TYPE ST_GetCamInfoParams :
STRUCT
  AtMasterPosition  : BOOL;
  MasterPosition    : LREAL;
END_STRUCT
END_TYPE

(* stored: Version 1.1.0.1, ProductVersion 3.1.4023.8
   DUT ST_GetCamInfoParams: Id {9b903223-9bde-487e-9d34-426d4bb37e27} *)
